Omron CX-Programmer project NewProject (CX-Programmer 9.61)

# PLC NewPLC1: CP1E E30

## Global symbols (name address type ; comment)
100.03 BOOL  ; motorFwd
100.04 BOOL  ; motorReverse
W10.00 BOOL  ; fwdSignal
W10.01 BOOL  ; stopSignal
W10.02 BOOL  ; revSignal
W20.00 BOOL  ; motorFwdSignal
W20.01 BOOL  ; motorRevSignal

## Program NewProgram1 (cyclic task 0)
; Forward Reverse motor with interlock
Local symbols
pilotLamp1 100.00 BOOL  ; PL1
pilotLamp2 100.01 BOOL
pilotLamp3 100.02 BOOL  ; PL3
pushButton1 0.00 BOOL
pushButton2 0.01 BOOL
pushButton3 0.02 BOOL

### Section Section1

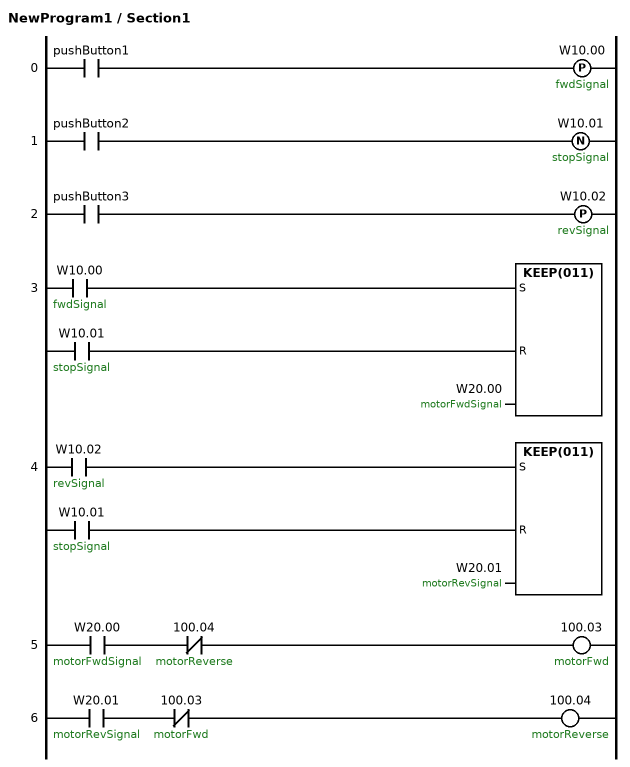
; rung 0
LD pushButton1
DIFU(013) W10.00  ; fwdSignal
; rung 1
LD pushButton2
DIFD(014) W10.01  ; stopSignal
; rung 2
LD pushButton3
DIFU(013) W10.02  ; revSignal
; rung 3
LD W10.00  ; fwdSignal
LD W10.01  ; stopSignal
KEEP(011) W20.00  ; motorFwdSignal
; rung 4
LD W10.02  ; revSignal
LD W10.01  ; stopSignal
KEEP(011) W20.01  ; motorRevSignal
; rung 5
LD W20.00  ; motorFwdSignal
ANDNOT 100.04  ; motorReverse
OUT 100.03  ; motorFwd
; rung 6
LD W20.01  ; motorRevSignal
ANDNOT 100.03  ; motorFwd
OUT 100.04  ; motorReverse

### Section END
; rung 0
END(001)